FUNCTION_BLOCK FB_EnableAxes
VAR_INPUT
	bEnableAxes: BOOL := TRUE;
END_VAR
VAR_OUTPUT
	bAllAxesReady: BOOL := FALSE;
END_VAR
VAR_IN_OUT
	io_X: AXIS_REF;
	io_Y: AXIS_REF;
	io_Z: AXIS_REF;
	io_C: AXIS_REF;
	io_M1: AXIS_REF;
	io_M2: AXIS_REF;
	io_M3: AXIS_REF;
	io_M4 : AXIS_REF;
END_VAR
VAR
	fOverride: LREAL := 100.0;
	fbPowerX: MC_Power;
	fbPowerY: MC_Power;
	fbPowerZ: MC_Power;
	fbPowerC: MC_Power;	
	fbPowerM1: MC_Power;
	fbPowerM2: MC_Power;
	fbPowerM3: MC_Power;
	fbPowerM4 : MC_Power;

END_VAR

io_X.ReadStatus();
io_Y.ReadStatus();
io_Z.ReadStatus();
io_C.ReadStatus();

io_M1.ReadStatus();
io_M2.ReadStatus();
io_M3.ReadStatus();
io_M4.ReadStatus();


fbPowerX(
	Enable:=bEnableAxes, 
	Enable_Positive:=bEnableAxes, 
	Enable_Negative:=bEnableAxes, 
	Override:=fOverride, 
	BufferMode:= , 
	Axis:=io_X, 
	Status=> , 
	Busy=> , 
	Active=> , 
	Error=> , 
	ErrorID=> );
fbPowerY(
	Enable:=bEnableAxes, 
	Enable_Positive:=bEnableAxes, 
	Enable_Negative:=bEnableAxes, 
	Override:=fOverride, 
	BufferMode:= , 
	Axis:=io_Y, 
	Status=> , 
	Busy=> , 
	Active=> , 
	Error=> , 
	ErrorID=> );	
fbPowerZ(
	Enable:=bEnableAxes, 
	Enable_Positive:=bEnableAxes, 
	Enable_Negative:=bEnableAxes, 
	Override:=fOverride, 
	BufferMode:= , 
	Axis:=io_Z, 
	Status=> , 
	Busy=> , 
	Active=> , 
	Error=> , 
	ErrorID=> );
fbPowerC(
	Enable:=bEnableAxes, 
	Enable_Positive:=bEnableAxes, 
	Enable_Negative:=bEnableAxes, 
	Override:=fOverride, 
	BufferMode:= , 
	Axis:=io_C, 
	Status=> , 
	Busy=> , 
	Active=> , 
	Error=> , 
	ErrorID=> );
	
	
fbPowerM1(
	Enable:=bEnableAxes, 
	Enable_Positive:=bEnableAxes, 
	Enable_Negative:=bEnableAxes, 
	Override:=fOverride, 
	BufferMode:= , 
	Axis:=io_M1, 
	Status=> , 
	Busy=> , 
	Active=> , 
	Error=> , 
	ErrorID=> );	
fbPowerM2(
	Enable:=bEnableAxes, 
	Enable_Positive:=bEnableAxes, 
	Enable_Negative:=bEnableAxes, 
	Override:=fOverride, 
	BufferMode:= , 
	Axis:=io_M2, 
	Status=> , 
	Busy=> , 
	Active=> , 
	Error=> , 
	ErrorID=> );	
fbPowerM3(
	Enable:=bEnableAxes, 
	Enable_Positive:=bEnableAxes, 
	Enable_Negative:=bEnableAxes, 
	Override:=fOverride, 
	BufferMode:= , 
	Axis:=io_M3, 
	Status=> , 
	Busy=> , 
	Active=> , 
	Error=> , 
	ErrorID=> );	
fbPowerM4(
	Enable:=bEnableAxes, 
	Enable_Positive:=bEnableAxes, 
	Enable_Negative:=bEnableAxes, 
	Override:=fOverride, 
	BufferMode:= , 
	Axis:=io_M4, 
	Status=> , 
	Busy=> , 
	Active=> , 
	Error=> , 
	ErrorID=> );
	
bAllAxesReady	:= fbPowerX.Status AND fbPowerY.Status AND fbPowerZ.Status AND fbPowerC.Status AND  
	fbPowerM1.Status AND fbPowerM2.Status AND fbPowerM3.Status AND fbPowerM4.Status;

END_FUNCTION_BLOCK

(* stored: Version 1.1.0.1, ProductVersion 3.1.4024.12
   POU FB_EnableAxes: Id {934bebd2-dcc5-45f7-9334-9a7406eb73c3}, SpecialFunc None *)
